KUKA KRL data list: ekxdemooriginal.dat

&ACCESS RVP
&PARAM TEMPLATE = C:\KRC\Roboter\Template\vorgabe
&PARAM EDITMASK = *
DEFDAT ekxdemooriginal
ENDDAT
